INTERFACE I_DatatypePack

METHOD RegisterWith
VAR_INPUT
	Datatypes : I_Datatypes;
END_VAR
END_METHOD

END_INTERFACE

(* stored: Version 1.1.0.1, ProductVersion 3.1.4024.12
   Itf I_DatatypePack: Id {e1cd5acd-cf5f-01e7-3ada-4a8d5051511e}
   Method RegisterWith: Id {a80882ed-4cbf-0b1c-2705-781730e52950} *)
